Universal Robots PolyScope program: cottonMachineOff.urp

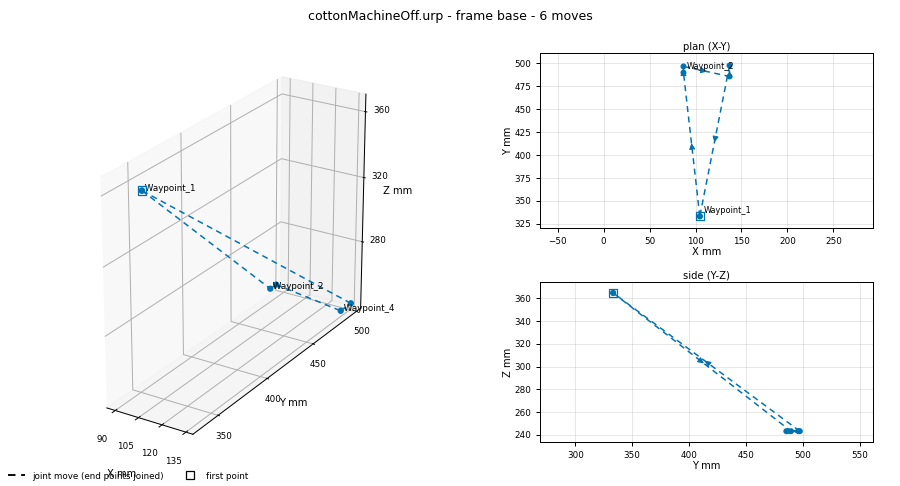
[picture p0: tool path of cottonMachineOff.urp in frame base, 6 of 8 moves have a stored position in this frame; points joined in program order, loops and branches not executed]
Program cottonMachineOff (installation=default directory=/programs/DavidMelin createdIn=5.12.4.1101661 lastSavedIn=5.12.4.1101661 robotSerialNumber=20225502378)
Calibrated DH parameters: a=[0.00022, -0.425328, -0.389701, 0.000059, 0.000065, 0]; d=[0.162608, 0.803456, 9.992211, -10.662202, 0.099702, 0.099559]; alpha=[1.570756, 0.001543, 0.004316, 1.570651, -1.570122, 0]; deltaTheta=[0, 0.002917, 0.116094, -0.119008, 0, -0.000001]
Robot Program (runOnlyOnce=true)
  MoveJ speed 60 deg/s, acceleration 80 deg/s^2 (useActiveTCP=true) feature=Base
    Waypoint Waypoint (Variable): variable=cotonHomePos
  URCap Gripper (Robotiq_Grippers, Robotiq Inc.) dataModel(position=100.0, force=0.0, speed=0.0, positionInDouble=100.0, forceInDouble=0.0, speedInDouble=0.0, slaveIds=[9], blocking=true)
  MoveJ speed 60 deg/s, acceleration 80 deg/s^2 (useActiveTCP=true) feature=Base
    Waypoint Waypoint_1: TCP in base x=104.654 y=333.279 z=364.791 mm, rx=-2.4906 ry=0.0958 rz=-0.1131 rad; joints [98.535, -64.728, -139.702, -29.678, 79.085, 9.451] deg
    Waypoint Waypoint_2: TCP in base x=86.868 y=489.697 z=243.23 mm, rx=-2.3949 ry=0.1183 rz=-0.0957 rad; joints [97.856, -105.116, -130.364, 6.938, 78.937, 9.481] deg
    Waypoint Waypoint_3: TCP in base x=86.861 y=496.459 z=243.237 mm, rx=-2.3949 ry=0.1183 rz=-0.0956 rad; joints [97.73, -105.82, -129.308, 6.606, 79.024, 9.385] deg
    Waypoint Waypoint_4: TCP in base x=136.995 y=485.535 z=243.217 mm, rx=-2.3949 ry=0.1184 rz=-0.0957 rad; joints [90.955, -106.171, -129.04, 7.482, 83.548, 4.286] deg
    Waypoint Waypoint_5: TCP in base x=136.99 y=497.448 z=243.216 mm, rx=-2.3949 ry=0.1184 rz=-0.0957 rad; joints [90.93, -107.352, -127.22, 6.845, 83.57, 4.268] deg
    Waypoint Waypoint_6: TCP in base x=104.648 y=333.283 z=364.786 mm, rx=-2.4906 ry=0.0958 rz=-0.1131 rad; joints [98.536, -64.728, -139.702, -29.678, 79.086, 9.452] deg
    Waypoint Waypoint (Variable): variable=cotonHomePos
